// TIA Portal V19 export
DATA_BLOCK "A0301_PERS"   // DB41
// stored: MemoryReserve 100
   VAR RETAIN
      Par : Struct
         Maint_FreeMove : Bool := FALSE;   // Manutenzione: movimento libero
         CaseA_PLen_Lim : Real := 700.0;   // [mm] Caso A : Lunghezza SG limite (da 900 a..)
         CaseA_StopperSensor : USInt := 1;   // Caso A : Sensori da usare su stopper
         CaseB_PLen_Lim : Real := 1990.0;   // [mm] Caso B : Lunghezza SG limite (da 900 a..)
         CaseB_StopperSensor : USInt := 3;   // Caso B : Sensori da usare su stopper
         CaseC_PLen_Lim : Real := 2000.0;   // [mm] Caso C : Lunghezza SG limite (da 900 a..)
         CaseC_StopperSensor : USInt := 3;   // Caso C : Sensori da usare su stopper
         CaseD_PLen_Lim : Real := 2100.0;   // [mm] Caso D : Lunghezza SG limite A (da 900 a..)
         CaseD_StopperSensor : USInt := 3;   // Caso D : Sensori da usare su stopper
         DlySensorsON { S7_SetPoint := 'True'} : Time := T#1S;   // [ms] Ritrado ON sensori prima e dopo fermi
         DlySensorsOFF { S7_SetPoint := 'True'} : Time := T#1S;   // [ms] Ritrado OFF sensori prima e dopo fermi
         TolReachNextStopper : Real := 70.0;   // [mm] Tolleranza movimento SG su stopper (Almeno un sensore in uso ON)
         TolReachAllSensorsON : Real := 50.0;   // [mm] Tolleranza posizione raggiunta (Sensori in uso ON)
      END_STRUCT;
      Par_Mng : Struct
         DlySensorsON { S7_SetPoint := 'True'} : Time := T#1S;   // [ms] Ritrado ON sensori prima e dopo fermi
         DlySensorsOFF { S7_SetPoint := 'True'} : Time := T#1S;   // [ms] Ritrado OFF sensori prima e dopo fermi
         TRK : Struct
            BTrk_MoveP4Exit { S7_SetPoint := 'True'} : Time := T#500MS;
            BTrk_MoveToP5 { S7_SetPoint := 'True'} : Time := T#500MS;
         END_STRUCT;
      END_STRUCT;
      Data_Mng { ExternalWritable := 'False'} : Struct
         LastCounter_PartMove_P2toP4 : LReal := 999999.999999998;
         LastCounter_PartMove_P1toP2 : LReal := 999999.999999998;
         LastCounter_PartMove_P1toP3 : LReal := 2.50784669856199;
      END_STRUCT;
   END_VAR
   VAR
      FC_Sensor : Struct
         "Case" : Int := 1;
      END_STRUCT;
   END_VAR
   VAR RETAIN
      SensTime : Struct
         P1 : Struct
            Sens_Ing : Struct
               DelayOn : Time := T#500MS;
            END_STRUCT;
            Sens_Out : Struct
               DelayOff : Time := T#300MS;
            END_STRUCT;
         END_STRUCT;
         P2 : Struct
            Sens_Ing : Struct
               DelayOn : Time := T#100MS;
            END_STRUCT;
            Sens_Out : Struct
               DelayOff : Time := T#500MS;
            END_STRUCT;
         END_STRUCT;
         P3 : Struct
            Sens_Ing : Struct
               DelayOn : Time := T#100MS;
            END_STRUCT;
            Sens_Out : Struct
               DelayOff : Time := T#100MS;
            END_STRUCT;
         END_STRUCT;
         P4 : Struct
            Sens_Ing : Struct
               DelayOn : Time := T#100MS;
            END_STRUCT;
            Sens_Out : Struct
               DelayOff : Time := T#100MS;
            END_STRUCT;
         END_STRUCT;
      END_STRUCT;
   END_VAR
BEGIN
END_DATA_BLOCK
